// TIA Portal V20 export
DATA_BLOCK "SP204"   // DB344
// stored: MemoryReserve 100
   VAR
      "MAIN OP EMERGENCY STOP CH.A" : Bool := TRUE;
      SPARE : Bool := FALSE;
      SPARE_1 : Bool := FALSE;
      SPARE_2 : Bool := FALSE;
      "MAIN OP EMERGENCY STOP CH.B" : Bool := FALSE;
   END_VAR
BEGIN
END_DATA_BLOCK
